Universal Robots PolyScope program: weigh_touch.urp

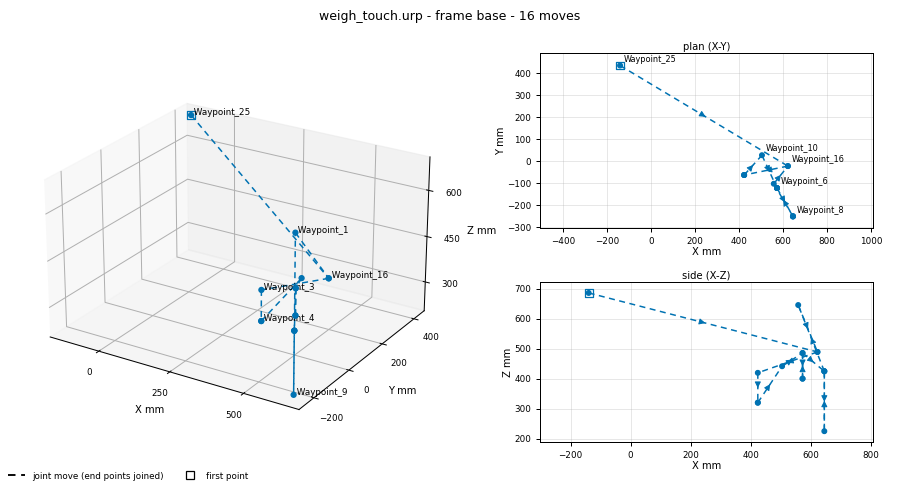
[picture p0: tool path of weigh_touch.urp in frame base, 16 of 16 moves have a stored position in this frame; points joined in program order, loops and branches not executed]
Program weigh_touch (installation=default directory=/programs/Nicolas_Arteaga/quality createdIn=5.8.2.10297 lastSavedIn=5.12.4.1101661 robotSerialNumber=20225502378)
Calibrated DH parameters: a=[0.00022, -0.425328, -0.389701, 0.000059, 0.000065, 0]; d=[0.162608, 0.803456, 9.992211, -10.662202, 0.099702, 0.099559]; alpha=[1.570756, 0.001543, 0.004316, 1.570651, -1.570122, 0]; deltaTheta=[0, 0.002917, 0.116094, -0.119008, 0, -0.000001]
Robot Program (runOnlyOnce=true)
  MoveJ speed 60 deg/s, acceleration 80 deg/s^2 (useActiveTCP=true) feature=Base
    Waypoint Waypoint_25: TCP in base x=-139.92 y=434.562 z=685.517 mm, rx=0.2728 ry=-1.6358 rz=-2.1043 rad; joints [228.521, -129.991, 99.843, -7.046, 27.223, 41.249] deg; TCP offset x=0 y=0 z=191.5 mm, rx=0 ry=0 rz=0 rad
    Waypoint Waypoint_16: TCP in base x=622.09 y=-21.999 z=488.949 mm, rx=0.729 ry=1.5781 rz=1.7949 rad; joints [135.515, -94.567, 106.176, -67.801, 9.2, 55.784] deg
    Waypoint Waypoint_3: TCP in base x=423.433 y=-62.575 z=419.467 mm, rx=-2.7081 ry=-1.5114 rz=-0.0978 rad; joints [150.374, -71.697, 50.193, 111.504, 85.496, 1.888] deg
    Waypoint Waypoint_4: TCP in base x=423.434 y=-62.603 z=320.013 mm, rx=-2.7081 ry=-1.5114 rz=-0.0977 rad; joints [150.402, -75.258, 69.862, 95.39, 85.495, 1.987] deg
    'Measure side 1 loop'
    Waypoint Waypoint_4: TCP in base x=423.434 y=-62.603 z=320.013 mm, rx=-2.7081 ry=-1.5114 rz=-0.0977 rad; joints [150.402, -75.258, 69.862, 95.39, 85.495, 1.987] deg
    Waypoint Waypoint_10: TCP in base x=504.298 y=27.412 z=441.351 mm, rx=-2.1458 ry=0.2085 rz=-0.4478 rad; joints [135.899, -74.63, 77.655, 112.181, 35.14, 43.687] deg
    Waypoint Waypoint_6: TCP in base x=572.488 y=-121.624 z=485.395 mm, rx=-1.4669 ry=0.8076 rz=-0.7838 rad; joints [121.615, -73.605, 85.33, 82.996, 2.356, 84.774] deg; TCP offset x=0 y=0 z=191.5 mm, rx=0 ry=0 rz=0 rad
    Waypoint Waypoint_7: TCP in base x=572.479 y=-121.672 z=400.008 mm, rx=-1.4669 ry=0.8075 rz=-0.784 rad; joints [121.623, -70.211, 93.438, 70.014, 2.368, 86.247] deg; TCP offset x=0 y=0 z=191.5 mm, rx=0 ry=0 rz=0 rad
    'measure height'
    Waypoint Waypoint_7: TCP in base x=572.479 y=-121.672 z=400.008 mm, rx=-1.4669 ry=0.8075 rz=-0.784 rad; joints [121.623, -70.211, 93.438, 70.014, 2.368, 86.247] deg
    Waypoint Waypoint_6: TCP in base x=572.488 y=-121.624 z=485.395 mm, rx=-1.4669 ry=0.8076 rz=-0.7838 rad; joints [121.615, -73.605, 85.33, 82.996, 2.356, 84.774] deg; TCP offset x=0 y=0 z=191.5 mm, rx=0 ry=0 rz=0 rad
    Waypoint Waypoint_8: TCP in base x=644.963 y=-250.234 z=424.745 mm, rx=-0.4223 ry=1.4905 rz=0.4378 rad; joints [121.021, -52.336, 61.566, 67.994, -2.525, 192.758] deg; TCP offset x=0 y=0 z=191.5 mm, rx=0 ry=0 rz=0 rad
    'measure side 2 loop'
    Waypoint Waypoint_8: TCP in base x=644.963 y=-250.234 z=424.745 mm, rx=-0.4223 ry=1.4905 rz=0.4378 rad; joints [121.021, -52.336, 61.566, 67.994, -2.525, 192.758] deg
    Waypoint Waypoint_9: TCP in base x=644.964 y=-250.243 z=224.998 mm, rx=-0.4223 ry=1.4905 rz=0.4378 rad; joints [121.04, -41.53, 74.294, 46.989, -2.465, 190.226] deg
    Waypoint Waypoint_8: TCP in base x=644.963 y=-250.234 z=424.745 mm, rx=-0.4223 ry=1.4905 rz=0.4378 rad; joints [121.021, -52.336, 61.566, 67.994, -2.525, 192.758] deg
    Waypoint Waypoint_1: TCP in base x=557.994 y=-102.204 z=645.214 mm, rx=-1.3174 ry=0.9174 rz=-0.5836 rad; joints [121.342, -85.625, 61.567, 24.73, -2.556, 192.757] deg
    Waypoint Waypoint_16: TCP in base x=622.09 y=-21.999 z=488.949 mm, rx=0.729 ry=1.5781 rz=1.7949 rad; joints [135.515, -94.567, 106.176, -67.801, 9.2, 55.784] deg
